// TwinCAT 3 PLC project PLC_daniel
// ProgramVersion: 3.1.4023.0
// libraries:
//   Tc2_Standard, * (Beckhoff Automation GmbH)
//   Tc2_System, * (Beckhoff Automation GmbH)
//   Tc3_Module, * (Beckhoff Automation GmbH)
// project tree:
//   Inputs/ Inputs.TcGVL
//   Inputs/Struct/ ST_AnalogInputStatus.TcDUT, ST_AnalogInput.TcDUT
//   Outputs/ Outputs.TcGVL
//   / PlcTask.TcTTO
//   POUs/ MAIN.TcPOU
// real-time tasks:
//   TASK PlcTask: cycle T#10ms, priority 20, ADS port 350
// I/O:
//   DEVICE PLC (EtherCAT), AmsNetId 5.80.90.242.2.1
//     PLC Rack (EK1200) [EK1200-5000 EtherCAT Power supply (2A E-Bus)]
//       DI (EL1008) [EL1008 8Ch. Dig. Input 24V, 3ms]
//       DO (EL2008) [EL2008 8Ch. Dig. Output 24V, 0.5A]
//       EndCap (EL9011) [EL9011 End Terminal]
//   DEVICE RIO (EtherCAT), AmsNetId 5.80.90.242.6.1
//     RIO Rack (EK1100) [EK1100 EtherCAT Coupler (2A E-Bus)]
//       DI (EL1008) [EL1008 8Ch. Dig. Input 24V, 3ms]
//       DO (EL2008) [EL2008 8Ch. Dig. Output 24V, 0.5A]
//       AI1 (EL3068) [EL3068 8Ch. Ana. Input 0-10V]
//       AI2 (EL3068) [EL3068 8Ch. Ana. Input 0-10V]
//       AI3 (EL3174) [EL3174 4Ch. Ana. Input +/-10V Diff., +/-20mA SingleEnded, 16 Bit]
//       AO (EL4104) [EL4104 4Ch. Ana. Output 0-10V, 16bit]
//       EndCap (EL9011) [EL9011 End Terminal]
// variable links:
//   PLC_daniel/PLC_daniel Instance <-> PLC (EtherCAT)/PLC Rack (EK1200)/DI (EL1008)
//     PlcTask Inputs/Inputs.bTest <-> Channel 1/Input
//   PLC_daniel/PLC_daniel Instance <-> PLC (EtherCAT)/PLC Rack (EK1200)/DO (EL2008)
//     PlcTask Outputs/Outputs.bTest <-> Channel 1/Output
//   PLC_daniel/PLC_daniel Instance <-> RIO (EtherCAT)/RIO Rack (EK1100)/AI1 (EL3068)
//     PlcTask Inputs/Inputs.stCylPos.nValue <-> AI Standard Channel 3/Value
//     PlcTask Inputs/Inputs.stCylPos.stStatus <-> AI Standard Channel 3/Status
//     PlcTask Inputs/Inputs.stJoyX.nValue <-> AI Standard Channel 1/Value
//     PlcTask Inputs/Inputs.stJoyX.stStatus <-> AI Standard Channel 1/Status
//     PlcTask Inputs/Inputs.stJoyY.nValue <-> AI Standard Channel 2/Value
//     PlcTask Inputs/Inputs.stJoyY.stStatus <-> AI Standard Channel 2/Status
//     PlcTask Inputs/Inputs.stSpoolPos.nValue <-> AI Standard Channel 4/Value
//     PlcTask Inputs/Inputs.stSpoolPos.stStatus <-> AI Standard Channel 4/Status
//   PLC_daniel/PLC_daniel Instance <-> RIO (EtherCAT)/RIO Rack (EK1100)/AI2 (EL3068)
//     PlcTask Inputs/Inputs.stFlowReturnSide.nValue <-> AI Standard Channel 7/Value
//     PlcTask Inputs/Inputs.stFlowReturnSide.stStatus <-> AI Standard Channel 7/Status
//     PlcTask Inputs/Inputs.stPressureCompensator.nValue <-> AI Standard Channel 3/Value
//     PlcTask Inputs/Inputs.stPressureCompensator.stStatus <-> AI Standard Channel 3/Status
//     PlcTask Inputs/Inputs.stPressureLhvSide.nValue <-> AI Standard Channel 5/Value
//     PlcTask Inputs/Inputs.stPressureLhvSide.stStatus <-> AI Standard Channel 5/Status
//     PlcTask Inputs/Inputs.stPressurePistonSide.nValue <-> AI Standard Channel 4/Value
//     PlcTask Inputs/Inputs.stPressurePistonSide.stStatus <-> AI Standard Channel 4/Status
//     PlcTask Inputs/Inputs.stPressureReturn.nValue <-> AI Standard Channel 2/Value
//     PlcTask Inputs/Inputs.stPressureReturn.stStatus <-> AI Standard Channel 2/Status
//     PlcTask Inputs/Inputs.stPressureRodSide.nValue <-> AI Standard Channel 6/Value
//     PlcTask Inputs/Inputs.stPressureRodSide.stStatus <-> AI Standard Channel 6/Status
//     PlcTask Inputs/Inputs.stPressureSupply.nValue <-> AI Standard Channel 1/Value
//     PlcTask Inputs/Inputs.stPressureSupply.stStatus <-> AI Standard Channel 1/Status
//   PLC_daniel/PLC_daniel Instance <-> RIO (EtherCAT)/RIO Rack (EK1100)/DI (EL1008)
//     PlcTask Inputs/Inputs.bAutoModeSelector <-> Channel 1/Input
//     PlcTask Inputs/Inputs.bManualModeSelector <-> Channel 2/Input
//     PlcTask Inputs/Inputs.bStartButton <-> Channel 3/Input
//     PlcTask Inputs/Inputs.bStopButton <-> Channel 4/Input
//   PLC_daniel/PLC_daniel Instance <-> RIO (EtherCAT)/RIO Rack (EK1100)/DO (EL2008)
//     PlcTask Outputs/Outputs.bGreenLight <-> Channel 1/Output
//     PlcTask Outputs/Outputs.bRedLight <-> Channel 2/Output

CONFIGURATION PLC_daniel
    RESOURCE PLC ON TwinCAT3
        TASK PlcTask(INTERVAL := T#10ms, PRIORITY := 20);
        PROGRAM MAIN WITH PlcTask : MAIN;
    END_RESOURCE
END_CONFIGURATION

// ---- Inputs/Struct/ST_AnalogInputStatus.TcDUT
TYPE ST_AnalogInputStatus :
STRUCT
	Underrange 		: BIT; // 0.0
	Overrange 		: BIT; // 0.1
	Limit_1_0 		: BIT; // 0.2
	Limit_1_1 		: BIT; // 0.3
	Limit_2_0 		: BIT; // 0.4
	Limit_2_1 		: BIT; // 0.5
	Error 			: BIT; // 0.6
	Reserved_0_7	: BIT; // 0.7
	Reserved_1_0 	: BIT; // 1.0
	Reserved_1_1 	: BIT; // 1.1
	Reserved_1_2 	: BIT; // 1.2
	Reserved_1_3 	: BIT; // 1.3
	Reserved_1_4 	: BIT; // 1.4
	Reserved_1_5 	: BIT; // 1.5
	TxPDO_State 	: BIT; // 1.6
	TxPDO_Toggle 	: BIT; // 1.7	
END_STRUCT
END_TYPE

// ---- Inputs/Struct/ST_AnalogInput.TcDUT
TYPE ST_AnalogInput :
STRUCT
	stStatus 	AT %I* : ST_AnalogInputStatus;
	nValue		AT %I* : INT;	
END_STRUCT
END_TYPE

// ---- Inputs/Inputs.TcGVL
{attribute 'qualified_only'}
VAR_GLOBAL
	
	// PLC Rack
	// Digital Inputs
	bTest 						AT %I* : BOOL;
	
	// RIO Rack
	// Digital Inputs
	bAutoModeSelector			AT %I* : BOOL;
	bManualModeSelector			AT %I* : BOOL;
	bStartButton				AT %I* : BOOL;
	bStopButton					AT %I* : BOOL;
	
	// Analog Inputs 1
	stJoyX 						: ST_AnalogInput;
	stJoyY						: ST_AnalogInput;
	stCylPos 					: ST_AnalogInput;
	stSpoolPos 					: ST_AnalogInput;
	
	// Analog Inputs 2
	stPressureSupply 			: ST_AnalogInput;
	stPressureReturn 			: ST_AnalogInput;
	stPressureCompensator 		: ST_AnalogInput;
	stPressurePistonSide 		: ST_AnalogInput;
	stPressureLhvSide 		    : ST_AnalogInput;
	stPressureRodSide			: ST_AnalogInput;
	
	// Analog Inputs 3 (Multi)
	stFlowReturnSide			: ST_AnalogInput;
END_VAR

// ---- Outputs/Outputs.TcGVL
{attribute 'qualified_only'}
VAR_GLOBAL
	// PLC Rack
	// Digital Outputs
	bTest					 AT %Q* : BOOL;
	
	// RIO Rack
	// Digital Outputs
	bGreenLight 			AT %Q* : BOOL;
	bRedLight 				AT %Q* : BOOL;
	// Analog Outputs
	nValveOutput 			AT %Q* : INT;
END_VAR

// ---- POUs/MAIN.TcPOU
PROGRAM MAIN
VAR
END_VAR

END_PROGRAM
